TYPE ST_ElapsedTime :
STRUCT
	Days		: INT;
	Hours		: INT;
	Minutes		: INT;
	Seconds		: INT;
END_STRUCT
END_TYPE

(* stored: Version 1.1.0.1, ProductVersion 3.1.4024.2
   DUT ST_ElapsedTime: Id {e3d73bcd-805f-4b2c-9fbb-4a840afbb2e8} *)
